PROGRAM MAIN
VAR
END_VAR

//******************************************
//cyclic call of all needed FB
//******************************************
ACT_Moteur();
ACT_Actor();

fbMMA();

//copy physical Inputs in fbBtn
fbBtn.xAru:=stio.stIn.IxAruIO;
fbBtn.xReset:=stio.stIn.xResetIO OR NOT stio.stIn.xAirPressureOk;
fbBtn.xStart:=stio.stIn.xStartIO;
fbBtn.xStop:=stio.stIn.xStopIO;
fbBtn.xAirPressureOk:=stio.stIn.xAirPressureOk;
fbBtn.xManualAct1GoIn:=stio.stIn.xManualAct1GoIn;
fbBtn.xManualAct1GoOut:=stio.stIn.xManualAct1GoOut;
fbBtn.xHomingPosReached:=stio.stIn.xHomingPosReached;
fbBtn.xSetHomePos:=stio.stIn.xSetHomePos;
fbBtn.xAllowedGetPiece:=stio.stIn.xAllowedGetPiece;
fbBtn.xPiecePresent:=stio.stIn.xPiecePresent;
fbBtn.xEmulateZDone:=stio.stIn.xEmulateZDone;
fbBtn.xJogXBackward:=stio.stIn.xJogXBackward;
fbBtn.xJogYBackward:=stio.stIn.xJogYBackward;
fbBtn.xJogXForward:=stio.stIn.xJogXForward;
fbBtn.xJogYForward:=stio.stIn.xJogYForward;
fbBtn.iMotorSpeed:=stio.stIn.iSetSpeedMotor;


//and now call it
fbBtn();

//stParam
//check for active errors
IF (fbAct1.stError.xState) THEN
	stParam.stStatus.xErreur:=TRUE;
	stParam.stStatus.iId:=fbAct1.stError.iId;
ELSIF (fbCycleAuto.xError) THEN
	stParam.stStatus.xErreur:=TRUE;
	stParam.stStatus.iId:=fbCycleAuto.iId;
ELSIF NOT fbBtn.xAirPressureOk THEN
	stParam.stStatus.xErreur:=TRUE;
	stParam.stStatus.iId:=1;
ELSE
	//clear the error State. Do not clear the last error Message to have some kind of error history
	stParam.stStatus.xErreur:=FALSE;
END_IF

//call auto mode and give over the needed parameters
fbCycleAuto.xStart:=fbMMA.iEtape=350;
fbCycleAuto.xStop:= fbMMA.iEtape=390;
fbCycleAuto.xReset:= fbMMA.iEtape=810 OR fbMMA.iEtape=910;
fbCycleAuto();

//call Init mode and give over the needed parameters
fbCycleInit.xStart:=(fbMMA.iEtape=110 OR fbMMA.iEtape=340);
fbCycleInit.xStop:= NOT (fbMMA.iEtape=111 OR fbMMA.iEtape=341);
fbCycleInit.xReset:= fbMMA.iEtape=810 OR fbMMA.iEtape=910;
fbCycleInit();
	
//call Manual mode and give over the needed parameters
fbCycleMan.xStart:= fbMMA.iEtape=210;
fbCycleMan.xStop:=  fbMMa.iEtape<>210;
fbCycleMan();


//******************************************
//Output actions
//******************************************

//activate Lamp1
stIo.stOut.QxLampeRed:=NOT fbBtn.xAru;

ACTION ACT_Actor:
//Air-Actor controlling part
//cyclic call of the FB-blocs
fbAct1();	//Act2 corresponds to taking the object

//actuator movement autorize only if not in ARU
fbAct1.xAutorizeIn:=fbBtn.xAru;
fbAct1.xAutorizeOut:=fbBtn.xAru;

//move in and out each actuator
fbAct1.xInGoOut:=fbCycleAuto.iEtape=113 OR fbCycleMan.iEtape=202;

fbAct1.xInGoIn:=fbCycleAuto.iEtape=180 OR fbCycleAuto.iEtape=122 OR fbCycleAuto.iEtape=150 OR fbCycleAuto.iEtape=800 OR fbCycleInit.iEtape=400 OR fbCycleMan.iEtape=201;

//Reset des Actionneurs avan le init
fbAct1.xReset:=fbCycleInit.iEtape=99 OR fbMMA.iEtape=810;
END_ACTION

ACTION ACT_Moteur:
//Motor controlling part
//exécution de l'appel du bloc moteur
fbMotorX(stParam:=stParam.stMachine.stParamMotX);
fbMotorY(stParam:=stParam.stMachine.stParamMotY);
fbMotorZ(stParam:=stParam.stMachine.stParamMotZ);


//pilotage mise en puissance
fbMotorX.mcPower.Enable:=stIO.stIn.IxAruIO;
fbMotorX.mcPower.Enable_Negative:=stIO.stIn.IxAruIO;
fbMotorX.mcPower.Enable_positive:=stIO.stIn.IxAruIO;
fbMotorX.mcPower.Override:=fbBtn.iMotorSpeed;
fbMotorX.mSetMoveAbsRapide();

fbMotorY.mcPower.Enable:=stIO.stIn.IxAruIO;
fbMotorY.mcPower.Enable_Negative:=stIO.stIn.IxAruIO;
fbMotorY.mcPower.Enable_positive:=stIO.stIn.IxAruIO;
fbMotorY.mcPower.Override:=fbBtn.iMotorSpeed;
fbMotorY.mSetMoveAbsLent();

fbMotorZ.mcPower.Enable:=stIO.stIn.IxAruIO;
fbMotorZ.mcPower.Enable_Negative:=stIO.stIn.IxAruIO;
fbMotorZ.mcPower.Enable_positive:=stIO.stIn.IxAruIO;
fbMotorZ.mcPower.Override:=fbBtn.iMotorSpeed;
fbMotorY.mSetMoveAbsLent();


//pilotage homing (prise d'origine)
fbMotorX.mcHome.Execute:=fbCycleInit.iEtape=100;
fbMotorX.mcHome.bCalibrationCam:=fbBtn.xHomingPosReached;

//pilotage homing (prise d'origine)
fbMotorY.mcHome.Execute:=fbCycleInit.iEtape=200;
fbMotorY.mcHome.bCalibrationCam:=fbBtn.xHomingPosReached;

//pilotage homing (prise d'origine)
fbMotorZ.mcHome.Execute:=fbCycleInit.iEtape=300;
fbMotorZ.mcHome.bCalibrationCam:=fbBtn.xHomingPosReached;


//pilotage Rest
fbMotorX.mcReset.Execute:=fbMMA.iEtape=810 OR fbCycleInit.iEtape=100;
fbMotorY.mcReset.Execute:=fbMMA.iEtape=810 OR fbCycleInit.iEtape=100;
fbMotorZ.mcReset.Execute:=fbMMA.iEtape=810 OR fbCycleInit.iEtape=100;

//pilotage déplacement absolu
fbMotorX.mcMoveAbsolute.Execute:=fbCycleAuto.iEtape=110 OR fbCycleAuto.iEtape=131;
fbMotorY.mcMoveAbsolute.Execute:=fbCycleAuto.iEtape=110 OR fbCycleAuto.iEtape=131;
fbMotorZ.mcMoveAbsolute.Execute:=fbCycleAuto.iEtape=112 OR fbCycleAuto.iEtape=120 OR fbCycleAuto.iEtape=141 OR fbCycleAuto.iEtape=161;

//Move Jog
fbMotorX.mcJog.JogForward:= fbBtn.xJogXForward AND (fbCycleInit.iEtape=500 OR fbCycleMan.iEtape=100);
fbMotorX.mcJog.JogBackwards:= fbBtn.xJogXBackward AND (fbCycleInit.iEtape=500 OR fbCycleMan.iEtape=100);
fbMotorY.mcJog.JogForward:= fbBtn.xJogYForward AND (fbCycleInit.iEtape=500 OR fbCycleMan.iEtape=100);
fbMotorY.mcJog.JogBackwards:= fbBtn.xJogYBackward AND (fbCycleInit.iEtape=500 OR fbCycleMan.iEtape=100);
END_ACTION

END_PROGRAM

(* stored: Version 1.1.0.1, ProductVersion 3.1.4020.12
   POU MAIN: Id {1e704377-3948-4a60-acf5-cdd6dbd4512e}, SpecialFunc None
   Action ACT_Actor: Id {414eda35-1edd-4eba-bf1d-081b5c6b8c4d}
   Action ACT_Moteur: Id {5fefa910-7333-41fc-b96a-1b2084cd9d5e} *)
